INTERFACE I_Session Extends I_Disposable

METHOD PUBLIC AddOrUpdateStorage
VAR_INPUT
	StorageId : T_MAXSTRING;
	Source : I_SessionData;
END_VAR
END_METHOD

METHOD PUBLIC DisposeAllDataFromStorage
VAR_INPUT
END_VAR
END_METHOD

METHOD PUBLIC DisposeDataFromStorage
VAR_INPUT
	StorageId : T_MAXSTRING;
END_VAR
END_METHOD

PROPERTY PUBLIC Id : T_MAXSTRING
GET
END_GET
END_PROPERTY

PROPERTY PUBLIC LastAccessedTimestamp : I_TimeStamp
GET
END_GET
END_PROPERTY

METHOD PUBLIC Refresh
VAR_INPUT
END_VAR
END_METHOD

METHOD PUBLIC TryGetDataFromStorage : BOOL
VAR_INPUT
	StorageId : T_MAXSTRING;
	Destination : REFERENCE TO I_SessionData;
END_VAR
END_METHOD

END_INTERFACE

(* stored: Version 1.1.0.1, ProductVersion 3.1.4026.13
   Itf I_Session: Id {02daf2cc-9508-444b-83cc-6a7ab37af681}
   Method AddOrUpdateStorage: Id {98d2f6bc-a3ae-4ab6-bec2-a17304829331}
   Method DisposeAllDataFromStorage: Id {5dc2f177-30e0-436a-ab62-ae041e2d8dbe}
   Method DisposeDataFromStorage: Id {d6d00990-b9c3-4623-944c-1ef8a0a570f9}
   Property Id: Id {27783e9f-f360-424f-9e88-8a4f5ba2ea72}
   Get Get: Id {94d53331-fbc2-41ad-9a8c-48e18c591513}
   Property LastAccessedTimestamp: Id {c1b2895b-984d-44a2-8ab5-c6f7750a8185}
   Get Get: Id {71b032c6-f00c-4f94-a7d6-0e752b063fb7}
   Method Refresh: Id {30ef096c-0925-4638-a02c-7fb641708fff}
   Method TryGetDataFromStorage: Id {4c1fc734-d03c-4264-aaf3-5d37b6bd5cc3} *)
